(* IEC 61131-3 sources: AXOpen/src/components.zebra.vision/ctrl/src/AxoEA3600/TypesStructuresAndEnums, 7 files *)

(* ---- eAxoEA3600BarcodeType.st ---- *)
NAMESPACE AXOpen.Components.Zebra.Vision
    TYPE PUBLIC
        eAxoEA3600BarcodeType : INT
        (
            none                                                    :=  0,
            Code_39                                                 :=  1,
            Codabar                                                 :=  2,
            Code_128                                                :=  3,
            Discrete_2_of_5_DTF                                     :=  4,
            IATA                                                    :=  5,
            Interleaved_2_of_5_ITF                                  :=  6,
            Code_93                                                 :=  7,
            UPC_A                                                   :=  8,
            UPC_E                                                   :=  9,
            EAN_8                                                   :=  10,
            EAN_13                                                  :=  11,
            Code_11                                                 :=  12,
            MSI                                                     :=  14,
            EAN_128                                                 :=  15,
            UPC_E1                                                  :=  16,
            PDF_417                                                 :=  17,
            Code_39_Full_ASCII_Conversion                           :=  19,
            Trioptic_Code_39                                        :=  21,
            Bookland_EAN                                            :=  22,
            UCC_Coupon_Extended_Code                                :=  23,
            ISBT_128                                                :=  25,
            MicroPDF417                                             :=  26,
            Data_Matrix                                             :=  27,
            QR_Code                                                 :=  28,
            US_Postnet                                              :=  30,
            US_Planet                                               :=  31,
            Code_32                                                 :=  32,
            ISBT_128_Concatenation                                  :=  33,
            Japan_Postal                                            :=  34,
            Australia_Post                                          :=  35,
            Netherlands_KIX_Code                                    :=  36,
            Maxicode                                                :=  37,
            UK_Postal                                               :=  39,
            Macro_PDF_417                                           :=  40,
            Micro_QR                                                :=  44,
            Aztec                                                   :=  45,
            GS1_DataBar_Omnidirectional_formerly_GS1_DataBar_14     :=  48,
            GS1_DataBar_Limited                                     :=  49,
            GS1_DataBar_Expanded                                    :=  50,
            USPS_4CB_One_Code_Intelligent_Mail                      :=  52,
            UPU_FICS_Postal                                         :=  53,
            ISSN_EAN                                                :=  54,
            Matrix_2_of_5                                           :=  57,
            UPCA_2                                                  :=  72,
            UPCE_2                                                  :=  73,
            EAN_8_2                                                 :=  74,
            EAN_13_2                                                :=  75,
            UPCE1_2                                                 :=  80,
            Composite_CC_A_EAN_128                                  :=  81,
            Composite_CC_A_EAN_13                                   :=  82,
            Composite_CC_A_EAN_8                                    :=  83,
            Composite_CC_A_RSS_Expanded                             :=  84,
            Composite_CC_A_RSS_Limited                              :=  85,
            Composite_CC_A_RSS_14                                   :=  86,
            Composite_CC_A_UPC_A                                    :=  87,
            Composite_CC_A_UPC_E                                    :=  88,
            Composite_CC_C_EAN_128                                  :=  89,
            TLC_39                                                  :=  90,
            Composite_CC_B_EAN_128                                  :=  97,
            Composite_CC_B_EAN_13                                   :=  98,
            Composite_CC_B_EAN_8                                    :=  99,
            Composite_CC_B_RSS_Expanded                             :=  100,
            Composite_CC_B_RSS_Limited                              :=  101,
            Composite_CC_B_RSS_14                                   :=  102,
            Composite_CC_B_UPC_A                                    :=  103,
            Composite_CC_B_UPC_E                                    :=  104,
            Chinese_2_of_5                                          :=  114,
            Korean_3_of_5                                           :=  115,
            GS1_Databar_Extended_Coupon                             :=  132,
            UPCA_5                                                  :=  136,
            UPCE_5                                                  :=  137,
            EAN_8_5                                                 :=  138,
            EAN_13_5                                                :=  139,
            UPCE1_5                                                 :=  144,
            GS1_Data_Matrix                                         :=  193,
            Han_Xin_Code                                            :=  183
        );
    END_TYPE
END_NAMESPACE

(* ---- AxoEA3600_Component_Status.st ---- *)
NAMESPACE AXOpen.Components.Zebra.Vision
    {S7.extern=ReadWrite}
    {#ix-attr:[Container(Layout.Stack)]}
    CLASS PUBLIC AxoEA3600_Component_Status EXTENDS AXOpen.Components.Abstractions.AxoComponent_Status
        VAR PUBLIC

        END_VAR
    END_CLASS
END_NAMESPACE

(* ---- AxoEA3600_Config.st ---- *)
NAMESPACE AXOpen.Components.Zebra.Vision
    {S7.extern=ReadWrite}
    {#ix-attr:[Container(Layout.Stack)]}
    CLASS PUBLIC AxoEA3600_Config
        VAR PUBLIC
            {#ix-set:AttributeName = "<#Info time#>"}
            InfoTime : LTIME := LT#5S;
            {#ix-set:AttributeName = "<#Error time#>"}
            ErrorTime : LTIME := LT#10S;
            {#ix-set:AttributeName = "<#Task timeout#>"}
            TaskTimeout : LTIME := LT#50S;
            {#ix-set:AttributeName = "<#Hardware IDs#>"}
            HWIDs : AxoEA3600_HWIDs;
            {#ix-set:AttributeName = "<#Enable handshake#>"}
            HandshakeEnable : BOOL := TRUE;   // Use ACK handshake
            {#ix-set:AttributeName = "<#Enable fragments#>"}
            FragmentEnable : BOOL := TRUE;   // Accept fragmented payloads (>64B)
            {#ix-set:AttributeName = "<#Continous reading#>"}
            ContinuousReading : BOOL := FALSE;
        END_VAR
    END_CLASS
END_NAMESPACE

(* ---- AxoEA3600_HWIDs.st ---- *)
NAMESPACE AXOpen.Components.Zebra.Vision
   {S7.extern=ReadWrite}
	CLASS AxoEA3600_HWIDs
      VAR PUBLIC
         {#ix-set:AttributeName = "<#Hardware ID  of the device#>"}
         HW_Device              :  UINT;
         {#ix-set:AttributeName = "<#Hardware ID of the 'BarcodeData_v2' submodule#>"}
         HwID_BarcodeData_v2            :   UINT;
      END_VAR
   END_CLASS
END_NAMESPACE

(* ---- AxoEA3600_In.st ---- *)
NAMESPACE AXOpen.Components.Zebra.Vision
    {S7.extern=ReadWrite}
    {#ix-attr:[Container(Layout.Wrap)]}
    CLASS PUBLIC AxoEA3600_In
        VAR PUBLIC
            {#ix-set:AttributeName = "<#Fragmented#>"}
            Status_Fragmented               :   BOOL;   // Set if barcode is fragmented
            {#ix-set:AttributeName = "<#First fragment#>"}
            Status_FirstFragment            :   BOOL;   // Set on first block of fragmented barcode
            {#ix-set:AttributeName = "<#Middle fragment#>"}
            Status_MiddleFragment           :   BOOL;   // Set on intermediate blocks of fragmented barcode
            {#ix-set:AttributeName = "<#Last fragment#>"}
            Status_LastFragment             :   BOOL;   // Set on last block of fragmented barcode
            {#ix-attr:[RenderIgnore()]}
            Status_Reserved_12              :   BOOL;   // Reserved / unused
            {#ix-attr:[RenderIgnore()]}
            Status_Reserved_13              :   BOOL;   // Reserved / unused
            {#ix-attr:[RenderIgnore()]}
            Status_Reserved_14              :   BOOL;   // Reserved / unused
            {#ix-attr:[RenderIgnore()]}
            Status_Reserved_15              :   BOOL;   // Reserved / unused
            {#ix-set:AttributeName = "<#Transfer enabled#>"}
            Status_TransferEnabled          :   BOOL;   // Set if barcode transfer is enabled
            {#ix-set:AttributeName = "<#Handshake enabled#>"}
            Status_HandshakeEnabled         :   BOOL;   // Set if transfer handshaking is enabled
            {#ix-set:AttributeName = "<#Fragmentation enabled#>"}
            Status_FragmentationEnabled     :   BOOL;   // Set if fragmentation of large barcodes is enabled
            {#ix-set:AttributeName = "<#Cache overflow#>"}
            Status_CacheOverflow            :   BOOL;   // Set if internal scanner cache overflows
            {#ix-set:AttributeName = "<#Input data overflow#>"}
            Status_InputDataOverflow        :   BOOL;   // Set if barcode data is larger than 494 bytes and is truncated
            {#ix-set:AttributeName = "<#Waiting for handshake#>"}
            Status_WaitingForHandshake      :   BOOL;   // Set if transfer is waiting for a handshake
            {#ix-set:AttributeName = "<#Trigger state#>"}
            Status_TriggerState             :   BOOL;   // Set when the trigger is pulled, cleared when released.
            {#ix-set:AttributeName = "<#Scanner type#>"}
            Status_ScannerType              :   BOOL;   // Reserved / unused
            {#ix-set:AttributeName = "<#Update counter#>"}
            UpdateCounter                   :   UINT;   // Incremented to indicate new barcode data
            {#ix-set:AttributeName = "<#Barcode type#>"}
            BarcodeType                     :   INT;    // Type of barcode contained in the Data field.
            {#ix-set:AttributeName = "<#Number of scanners#>"}
            NumberOfAttachedScanners        :   BYTE;
            {#ix-set:AttributeName = "<#Battery charge state#>"}
            BatteryStateOfCharge            :   BYTE;
            {#ix-set:AttributeName = "<#Battery voltage#>"}
            BatteryVoltage                  :   INT;
            {#ix-set:AttributeName = "<#Battery temperature#>"}
            BatteryTemp                     :   INT;
            {#ix-attr:[RenderIgnore()]}
            BatteryDateOfManufacture        :   ARRAY[0..7] OF BYTE;    // Reserved for future expansion
            {#ix-attr:[RenderIgnore()]}
            Reserved                        :   INT;
            {#ix-set:AttributeName = "<#Length of the data#>"}
            Length                          :   UINT;   // Length of barcode data in the Data field
            Data                            :   ARRAY[0..63] OF BYTE;   // Barcode data
        END_VAR
    END_CLASS
END_NAMESPACE

(* ---- AxoEA3600_Out.st ---- *)
NAMESPACE AXOpen.Components.Zebra.Vision
    {S7.extern=ReadWrite}
    {#ix-attr:[Container(Layout.Wrap)]}
    CLASS PUBLIC AxoEA3600_Out
        VAR PUBLIC
            Ctrl_Reserved_8             : BOOL;   // Reserved / unused
            Ctrl_Reserved_9             : BOOL;   // Reserved / unused
            Ctrl_Reserved_10            : BOOL;   // Reserved / unused
            Ctrl_Reserved_11            : BOOL;   // Reserved / unused
            Ctrl_Reserved_12            : BOOL;   // Reserved / unused
            Ctrl_Reserved_13            : BOOL;   // Reserved / unused
            Ctrl_Reserved_14            : BOOL;   // Reserved / unused
            Ctrl_Reserved_15            : BOOL;   // Reserved / unused
            Ctrl_EnableTransfer         : BOOL;   // Set to enable barcode transfer
            Ctrl_EnableHandshake        : BOOL;   // Set to enable transfer handshaking
            Ctrl_EnableFragmentation    : BOOL;   // Set to enable fragmentation of large barcodes
            Ctrl_Reserved_3             : BOOL;   // Reserved / unused
            Ctrl_ClearFaults            : BOOL;   // Set to clear faults in the scanner barcode transfer interface
            Ctrl_StartScan              : BOOL;   // Set to start scan session.
            Ctrl_StopScan               : BOOL;   // Set to stop scan session.
            Ctrl_SendAction             : BOOL;   // Set to trigger the scanner user action.
            AckCounter                  : UINT;   // Used in transfer handshaking to indicate that the data block has been processed
            UIActionCode                : WORD;   // Scanner user indication code
        END_VAR
    END_CLASS
END_NAMESPACE

(* ---- AxoEA3600_ReadData.st ---- *)
NAMESPACE AXOpen.Components.Zebra.Vision
    {S7.extern=ReadWrite}
    CLASS PUBLIC AxoEA3600_ReadData EXTENDS AXOpen.Core.AxoByteArray
        VAR PUBLIC
            Data : ARRAY [0..1023] OF BYTE;
        END_VAR
    END_CLASS
END_NAMESPACE
